Yaskawa INFORM job: DUMMY_PAINT.JBI

/JOB
//NAME DUMMY_PAINT
//POS
///NPOS 1,0,0,0,0,0
///TOOL 0
///POSTYPE PULSE
///PULSE
C00000=48311,124721,-96380,117016,-92698,-15405
//INST
///DATE 2022/12/26 14:59
///ATTR SC,RW
///GROUP1 RB1
NOP
MOVJ C00000 VJ=15.00
SPYON
SPYOF
END
